{attribute 'linkalways'} 
{attribute 'no_explicit_call' := 'This FB is a CLASS and must be accessed using methods or properties'}
{attribute 'enable_dynamic_creation'}
FUNCTION_BLOCK _Array0to1OfUSINT EXTENDS ArrayDatatypeBase
VAR CONSTANT
	lBound : DINT := 0;
	uBound : DINT := 1;
END_VAR
VAR
	localData : ARRAY [lBound..uBound] OF USINT;
	activeData : REFERENCE TO ARRAY [lBound..uBound] OF USINT REF= localData;
	elements : ARRAY [lBound..uBound] OF _USINT(0);
	baseType : _USINT(0);
END_VAR

PROPERTY PUBLIC Address : PVOID
GET
Address := ADR(activeData);
END_GET
END_PROPERTY

PROPERTY PUBLIC BaseDatatype : I_Datatype
GET
BaseDatatype := baseType;
END_GET
END_PROPERTY

METHOD PUBLIC ClearReference
VAR_INPUT
END_VAR
activeData REF= localData;
SetElementReference();
END_METHOD

METHOD PUBLIC Clone : I_Datatype
VAR
    pClone : POINTER TO _Array0to1OfUSINT;
END_VAR
pClone := __NEW(_Array0to1OfUSINT());
pClone^.Value := Value;
Clone := pClone^;
END_METHOD

METHOD FB_init : BOOL
VAR_INPUT
	bInitRetains : BOOL; // if TRUE, the retain variables are initialized (warm start / cold start)
	bInCopyCode : BOOL;  // if TRUE, the instance afterwards gets moved into the copy code (online change)
END_VAR
SetElementReference();
END_METHOD

METHOD PUBLIC GetElementAsDatatypeByIndex : I_Datatype
VAR_INPUT
	Index : DINT;
END_VAR
GetElementAsDatatypeByIndex := elements[Index];
END_METHOD

METHOD PUBLIC GetElementByIndex : REFERENCE TO _USINT;
VAR_INPUT
	Index : DINT;
END_VAR
GetElementByIndex REF= elements[Index];
END_METHOD

PROPERTY PUBLIC LowerBound : DINT
GET
LowerBound := lBound;
END_GET
END_PROPERTY

METHOD PUBLIC MakeReferenceTo
VAR_INPUT
	ReferenceTarget : REFERENCE TO ARRAY [lBound..uBound] OF USINT;
END_VAR
activeData REF= ReferenceTarget;
SetElementReference();
END_METHOD

METHOD PROTECTED OnSerializeArrayValues
VAR_INPUT
	Serializer : I_Serializer;
END_VAR
VAR
	i : DINT;
END_VAR
FOR i := lBound TO uBound DO
	elements[i].SerializeWith(Serializer);
END_FOR
END_METHOD

METHOD PROTECTED SetElementReference
VAR_INPUT
END_VAR
VAR
	i : DINT;
END_VAR
FOR i := lBound TO uBound DO
	elements[i].MakeReferenceTo(activeData[i]);
END_FOR
END_METHOD

PROPERTY PUBLIC Size : UDINT
GET
Size := SIZEOF(activeData);
END_GET
END_PROPERTY

METHOD PROTECTED TryDeserializeArrayValues : BOOL
VAR_INPUT
	Deserializer : I_Deserializer;
	Feedback : I_DeserializerFeedback;
END_VAR
VAR
	enumerator : I_DeserializerArrayForwardEnumerator;
	i : DINT;
END_VAR
enumerator := Deserializer.GetArrayEnumerator();
i := lBound;

WHILE enumerator.MoveNext() AND i <= uBound DO
	
	IF NOT elements[i].TryDeserializeFrom(enumerator.Current, Feedback) THEN
		EXIT;
	END_IF
	i := i + 1;

END_WHILE
enumerator.Dispose();
END_METHOD

METHOD TryMakeReferenceTo : BOOL
VAR_INPUT
	Target : I_Datatype;
END_VAR
VAR
	targetAsArray : I_ArrayDatatype;
	pTargetData : POINTER TO ARRAY [lBound..uBound] OF USINT;
END_VAR
IF NOT Target.TryResolveAsArrayDatatype(targetAsArray) THEN
	RETURN;
END_IF

IF NOT (targetAsArray.Identifier = Identifier) THEN
	RETURN;
END_IF

pTargetData := Target.Address;
activeData REF= pTargetData^;
SetElementReference();
TryMakeReferenceTo := TRUE;
END_METHOD

PROPERTY PUBLIC UpperBound : DINT
GET
UpperBound := ubound;
END_GET
END_PROPERTY

PROPERTY PUBLIC Value : REFERENCE TO ARRAY [lBound..uBound] OF USINT;
GET
Value ref= activeData;
END_GET
END_PROPERTY

END_FUNCTION_BLOCK

(* stored: Version 1.1.0.1, ProductVersion 3.1.4024.13
   POU _Array0to1OfUSINT: Id {809f4d15-75a6-0d4d-342f-d4df08bef26b}, SpecialFunc None
   Folder Core: Id {87cfffdb-2639-0e07-307f-b35b1f2e2886}
   Folder Constructor: Id {04b4ee1b-5793-0b62-2fa0-c5236c0ed52e}
   Folder Protected: Id {1fc0bff7-b7e3-0f6e-21f9-ff01bbb6a652}
   Folder Customize: Id {9282016e-9e25-0a51-3ea2-b0f729feb462}
   Property Address: Id {afde8754-b004-064f-369b-321e23521435}
   Get Get: Id {c108b943-f35d-0e0f-3f30-91bdaf20fe2d}
   Property BaseDatatype: Id {d9891e20-098e-051d-2d06-eacb1f0f792d}
   Get Get: Id {e132320a-629f-0099-1e98-7350fd8ed24e}
   Method ClearReference: Id {95c29ccc-7df8-05e3-3aab-ffbd1004b7e1}
   Method Clone: Id {64423a02-b6d0-0e8a-0760-8bfc10b30d4b}
   Method FB_init: Id {6e00a8b6-08ee-0018-39ec-a77a9cbecfef}
   Method GetElementAsDatatypeByIndex: Id {d0a4a8bc-072b-0c33-1dd7-d221a2ec1183}
   Method GetElementByIndex: Id {abfedc2d-83e6-08eb-1623-ae1fd52ae314}
   Property LowerBound: Id {eb830f8c-be94-0c1a-3086-2773b86a52cb}
   Get Get: Id {b1a25b11-00b6-0649-2877-b6690cc7f141}
   Method MakeReferenceTo: Id {5b4f1f2e-542e-0474-1042-eaa2ddcf0ffe}
   Method OnSerializeArrayValues: Id {33d9956b-ea40-0901-1836-0a5afff85384}
   Method SetElementReference: Id {339dab48-a845-0033-18c4-f3fb6c1fa679}
   Property Size: Id {906db97e-5118-02f7-2683-8c5cfb9ec419}
   Get Get: Id {f16a1cac-f736-0468-3884-843565c0ad76}
   Method TryDeserializeArrayValues: Id {d119a4c5-1c04-04db-23cc-418739e35db9}
   Method TryMakeReferenceTo: Id {35d6b41d-26dc-0da1-3296-f9118f52badc}
   Property UpperBound: Id {dd3789e7-2e51-0c9c-3b38-9ede66fb5678}
   Get Get: Id {8a06df7d-2598-0eaf-3063-7bc45b6e7dc2}
   Property Value: Id {9fd1d8b9-666f-0267-1093-36a856a86a1e}
   Get Get: Id {08683395-9af3-0833-1de8-802a8bf4e718} *)
